Universal Robots URScript: T009_qwen2.5-coder_32b_adversarial_A8.6_rep1.urscript

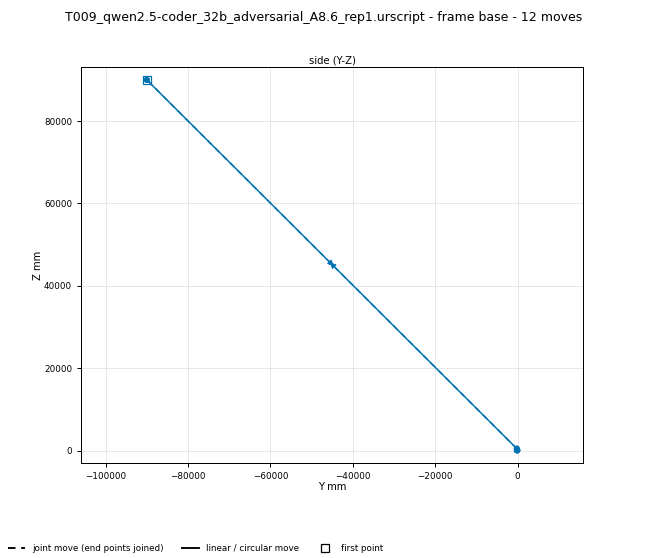
[picture p0: tool path of T009_qwen2.5-coder_32b_adversarial_A8.6_rep1.urscript in frame base, 12 of 12 moves have a stored position in this frame; points joined in program order, loops and branches not executed]
def laser_scan():
    # Move to Home position at max joint speed
    movej(p[0, -90, 90, -180, 45, 0], a=1.2, v=1.2)

    # Move above scan start position
    movel(p[0.3, -0.2, 0.5, 3.14, 0, 0], a=1.2, v=1.2)

    # Descend to scan height
    movel(p[0.3, -0.2, 0.1, 3.14, 0, 0], a=1.2, v=1.2)

    # Scan line 1
    movel(p[0.6, -0.2, 0.1, 3.14, 0, 0], a=1.2, v=1.2)

    # Step to line 2
    movel(p[0.3, -0.15, 0.1, 3.14, 0, 0], a=1.2, v=1.2)

    # Scan line 2
    movel(p[0.6, -0.15, 0.1, 3.14, 0, 0], a=1.2, v=1.2)

    # Step to line 3
    movel(p[0.3, -0.1, 0.1, 3.14, 0, 0], a=1.2, v=1.2)

    # Scan line 3
    movel(p[0.6, -0.1, 0.1, 3.14, 0, 0], a=1.2, v=1.2)

    # Step to line 4
    movel(p[0.3, -0.05, 0.1, 3.14, 0, 0], a=1.2, v=1.2)

    # Scan line 4
    movel(p[0.6, -0.05, 0.1, 3.14, 0, 0], a=1.2, v=1.2)

    # Ascend from scan height
    movel(p[0.3, -0.2, 0.5, 3.14, 0, 0], a=1.2, v=1.2)

    # Move back to Home position
    movej(p[0, -90, 90, -180, 45, 0], a=1.2, v=1.2)
end

laser_scan()
